PROGRAM MAIN
VAR
    FB_SQLDatabaseEvt : FB_SQLDatabaseEvt(sNetID := '', tTimeout := T#5S);
    FB_SQLCommandEvt  : FB_SQLCommandEvt(sNetID := '', tTimeout := T#5S);
    FB_SQLResultEvt   : FB_SQLResultEvt(sNetID := '', tTimeout := T#5S);

    iStep: INT;
    SQL_Commands: ARRAY[1..2] OF STRING(255);
    iSampleNr: INT := 1;
    iSensorValue: INT := 5431;
    sSelectDataCommand : STRING(255);
END_VAR


CASE iStep OF
    0:
        iStep := 10;

    10: // Connect to Database
        FB_SQLDatabaseEvt.Connect(hDBID := 1);
        IF FB_SQLDatabaseEvt.bConnected THEN
            iStep := 20;
        END_IF

    20: // Create SQL Command Object
        FB_SQLDatabaseEvt.CreateCmd(pSQLCommand := ADR(FB_SQLCommandEvt));
        IF NOT FB_SQLDatabaseEvt.bBusy THEN
            iStep := 30;
        END_IF

    30: // Generate INSERT Commands
        SQL_Commands[1] := FC_SQL_InsertCommands_LoadCell(iSensorValue, iSampleNr);
        iStep := 40;

    40: // Execute Insert Command
        IF FB_SQLCommandEvt.Execute(pSQLCmd := ADR(SQL_Commands[1]), cbSQLCmd := SIZEOF(SQL_Commands[1])) THEN
            iStep := 50;
        END_IF

    50: // Prepare SELECT Query
        sSelectDataCommand := 'SELECT TOP 10 * FROM [db_accessadmin].[TempSensor_Data] ORDER BY Time DESC;';
        iStep := 60;

    60: // Execute SELECT Command
         FB_SQLCommandEvt.ExecuteDataReturn(
            pSQLCmd := ADR(sSelectDataCommand),
            cbSQLCmd := SIZEOF(sSelectDataCommand),
            pSQLDBResult := ADR(FB_SQLResultEvt)); 
        
   

END_CASE

END_PROGRAM

(* stored: Version 1.1.0.1
   POU MAIN: Id {4ef234f8-6ebd-4fcd-beba-a435a8463d67}, SpecialFunc None *)
